(* PLC project Generated.project, CODESYS CODESYS V3.5 SP19 Patch 1 *)
(* stored: creationDateTime 2026-09-06T13:00:42.548374, modificationDateTime 2026-09-06T13:00:42.548374 *)

TYPE ST_ChainContextGlobal : STRUCT
  Idx101_ModeActive : E_Mode;  (* Mode de marche actif (MANUEL, SEMI_AUTO, MAINT_N1, MAINT_N2) *)
  Idx102_SimulationEnabled : BOOL;  (* 0 = Matériel Réel (Nominal) | 1 = SIMULATION ACTIVE ⚠️ *)
  Idx103_JoystickCommOk : BOOL;  (* 1 = Comm CANopen Joystick OK (Sain) | 0 = Perte Comm CAN *)
  Idx201_JoystickSelected : BOOL;  (* 1 = Pilotage par Joystick Hall | 0 = Pilotage par Boutons IHM *)
  Idx202_BypassNetworkGlobal : BOOL;  (* 0 = Comm Réseau OK | 1 = BYPASS RÉSEAU ACTIF ⚠️ *)
  Idx203_BypassSensorsGlobal : BOOL;  (* 0 = Capteurs Actifs | 1 = AU MOINS 1 CAPTEUR SHUNTÉ ⚠️ *)
  Idx301_EmergencyChainClosed : BOOL;  (* 1 = Boucle AU Matérielle Fermée (OK) | 0 = AU APPUYÉ *)
  Idx302_PowerContactorEngaged : BOOL;  (* 1 = Puissance Armée | 0 = Puissance Coupée *)
  Idx303_SafeStopActiveAny : BOOL;  (* 0 = Sain | 1 = AU MOINS UN SAFESTOP MÉTIER ACTIF *)
  Idx304_PowerCutOffActiveAny : BOOL;  (* 0 = Sain | 1 = COUPURE GENERAL COLLAGE ACTIVEE *)
  Idx401_HmiHeartbeatOk : BOOL;  (* 1 = Liaison IHM Active | 0 = Perte Liaison IHM *)
  Idx402_CycleAutoBusy : BOOL;  (* 1 = Séquenceur Auto en Cours | 0 = Repos *)
END_STRUCT;
END_TYPE

(* values of E_Mode: DISABLE: Mode Désactivé / Veille de sécurité (sorties bloquées); MAINT_N1: Manuel Niveau 1 : Pilotage unitaire avec toutes sécurités actives; MAINT_N2: Manuel Niveau 2 : Pilotage dégradé (droits étendus + bypasses autorisés); SEMI_AUTO: Mode Semi-Automatique (séquenceur automatique) *)

{attribute 'qualified_only'}
{attribute 'strict'}
TYPE E_Mode : (DISABLE := 0, MAINT_N1 := 1, MAINT_N2 := 2, SEMI_AUTO := 3);
END_TYPE
